PROGRAM MAIN
VAR
END_VAR

END_PROGRAM

(* stored: Version 1.1.0.1, ProductVersion 3.1.0.36
   POU MAIN: Id {e7f94cbd-a88e-4959-bea0-6e0449aa4fb2} *)
